// Writes a fixed64 field value, without a tag, to the stream.
FUNCTION F_WriteFixed64 : HRESULT
VAR_IN_OUT
    aBuffer : ARRAY [*] OF BYTE;
    stState : ST_WriterInternalState;
END_VAR
VAR_INPUT
    nValue : ULINT;
END_VAR
VAR
END_VAR

F_WriteFixed64 := F_WriteRawLittleEndian64(aBuffer, stState, nValue);

END_FUNCTION

(* stored: Version 1.1.0.1
   POU F_WriteFixed64: Id {51775a41-adec-4d53-a0bc-e99ec47dceec}, SpecialFunc None *)
